(* PLC project BACnet, Unknown Unnamed 1 *)
(* stored: creationDateTime 2018-07-28T02:24:08, modificationDateTime 2018-07-29T01:54:59 *)

FUNCTION_BLOCK Simulator
  VAR_OUTPUT
    Out : REAL;
  END_VAR
  VAR_INPUT
    MinVal : REAL;
    MaxVal : REAL;
    PeriodSeconds : INT;
  END_VAR
  VAR
    TON0 : TON;
    seconds : INT;
    BaseVal : REAL;
    VarVal : REAL;
  END_VAR

            (* pseudo-random variations *)
TON0(IN := TRUE, PT := T#3120s);
IF TON0.Q THEN
  TON0(IN := FALSE);
END_IF;
seconds := TIME_TO_INT(TON0.ET);

BaseVal := (MaxVal + MinVal)/2.0;
VarVal  := (MaxVal-MinVal)*INT_TO_REAL((seconds MOD PeriodSeconds) - (PeriodSeconds/2))/INT_TO_REAL(PeriodSeconds);

Out :=  BaseVal + VarVal;
          
END_FUNCTION_BLOCK

PROGRAM program0
  VAR
    EnergyCounter AT %MD0.2.0 : REAL;
    Temperature AT %ID0.0.0 : REAL;
    Humidity AT %ID0.0.1 : REAL;
  END_VAR
  VAR
    TempSimulation : Simulator;
    HumiditySimulation : Simulator;
  END_VAR
  VAR
    TemperatureSetPoint AT %QD0.1.0 : REAL;
    ControlDisable AT %QX0.4.2 : BOOL;
    Heater AT %IX0.3.0 : BOOL;
    Cooler AT %IX0.3.1 : BOOL;
  END_VAR

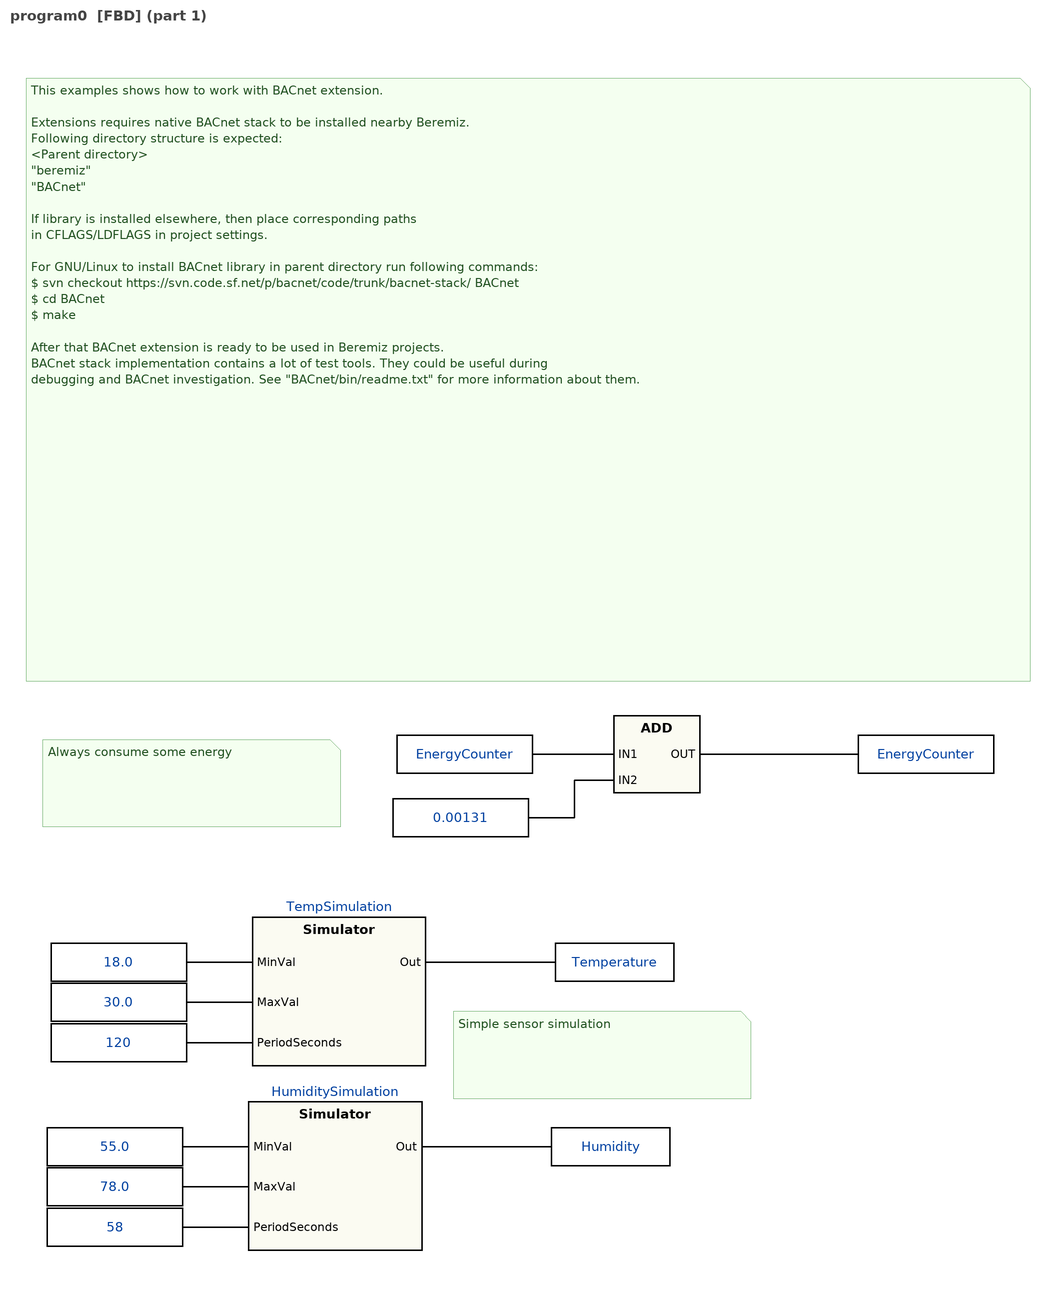
(* FBD diagram, written out as Structured Text *)
(* This examples shows how to work with BACnet extension.

Extensions requires native BACnet stack to be installed nearby Beremiz.
Following directory structure is expected:
<Parent directory>
  "beremiz"
  "BACnet"

If library is installed elsewhere, then place corresponding paths
in CFLAGS/LDFLAGS in project settings.

For GNU/Linux to install BACnet library in parent directory run following commands:
$ svn checkout https://svn.code.sf.net/p/bacnet/code/trunk/bacnet-stack/ BACnet
$ cd BACnet
$ make

After that BACnet extension is ready to be used in Beremiz projects.
BACnet stack implementation contains a lot of test tools. They could be useful during 
debugging and BACnet investigation. See "BACnet/bin/readme.txt" for more information about them. *)
(* Always consume some energy *)
EnergyCounter := EnergyCounter + 0.00131;
TempSimulation(MinVal := 18.0, MaxVal := 30.0, PeriodSeconds := 120);
Temperature := TempSimulation.Out;
(* Simple sensor simulation *)
HumiditySimulation(MinVal := 55.0, MaxVal := 78.0, PeriodSeconds := 58);
Humidity := HumiditySimulation.Out;
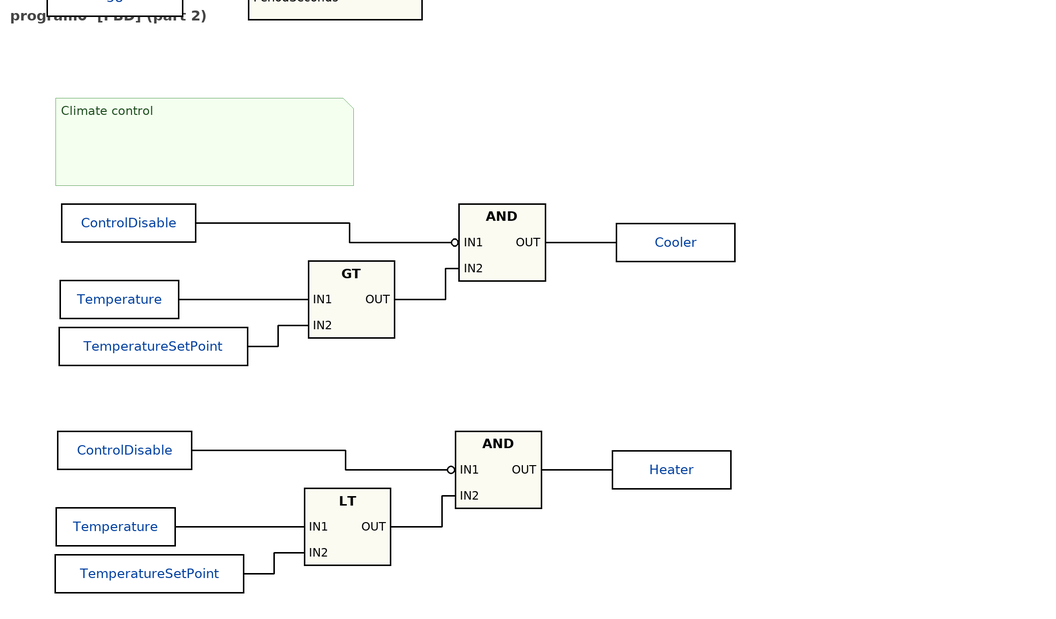
(* Climate control *)
Cooler := NOT ControlDisable AND Temperature > TemperatureSetPoint;
Heater := NOT ControlDisable AND Temperature < TemperatureSetPoint;
END_PROGRAM

CONFIGURATION config
  RESOURCE resource1 ON PLC
    TASK task0(INTERVAL := T#20ms, PRIORITY := 0);
    PROGRAM instance0 WITH task0 : program0;
  END_RESOURCE
END_CONFIGURATION
